FUNCTION_BLOCK Cylinder EXTENDS A_Actuator
VAR_INPUT
	
END_VAR
VAR_OUTPUT
	bExtended : BOOL;
	bExtend : BOOL;
END_VAR
VAR
	fbExtendedSignal : BoolIn;
	fbExtend : BoolOut;
END_VAR

super^();

bExtended := fbExtendedSignal.getValue;
bExtend := fbExtend.getValue;

METHOD  executeCmd : BOOL
VAR_INPUT
	
END_VAR
SUPER^.executeCmd();

CASE eCmd OF
	ePUSH:
		extend();
	eRETRACT:
		retract();
END_CASE
END_METHOD

METHOD extend : BOOL
VAR_INPUT
END_VAR
fbExtend.setValue := TRUE;
END_METHOD

PROPERTY getExtend : I_StepCondition
GET
getExtend := fbExtend;
END_GET
END_PROPERTY

METHOD retract : BOOL
VAR_INPUT
END_VAR
fbExtend.setValue := FALSE;
END_METHOD

END_FUNCTION_BLOCK

(* stored: Version 1.1.0.1, ProductVersion 3.1.4024.2
   POU Cylinder: Id {4dff6417-8bf1-4724-a444-43bb6b5867e9}, SpecialFunc None
   Method executeCmd: Id {23506408-3588-4191-8f91-d0bdab62d4fc}
   Method extend: Id {959ae6c2-4214-4061-b579-5b43c63e1617}
   Property getExtend: Id {551c2e8d-9793-498c-9e33-32fe5f29706c}
   Get Get: Id {70090b27-bd92-4955-9176-2f006b2ffbdc}
   Method retract: Id {8f00f682-12a1-4f93-aad1-7d8e6b2d1427} *)
